KUKA KRL data list: UP1.dat

&ACCESS RVP
&REL 1
&COMMENT Auto-loop PTP Move to P1 with external trigger
DEFDAT SIMPLE_MOVE

; Define position P1
DECL E6POS P1={x 309.227112,y -149.653107,z 1745.69702,a -77.6270523,b -57.8837891,c -160.023407,s 2,t 34,e1 0.0,e2 0.0,e3 0.0,e4 0.0,e5 0.0,e6 0.0}

ENDDAT
